KUKA KRL program: TORQUE.src

&ACCESS RV
&REL 9
&PARAM TEMPLATE = C:\KRC\Roboter\Template\FunctionVorgabe
&PARAM EDITMASK = *
DEFFCT BOOL TORQUE( )
DECL FRAME PT1
$TOOL=TOOL_DATA[5]
$ORI_TYPE=#CONSTANT
$VEL.CP=1.0
$VEL.ORI1=100
$VEL.ORI2=100
$ACC.CP=1.0
$ACC.ORI1=100
$ACC.ORI2=100

PTP $AXIS_ACT
IF $POS_ACT.A > 0 THEN
PTP_REL {A -1}
ENDIF
IF $POS_ACT.A < 0 THEN
PTP_REL {A 1}
ENDIF


ENDFCT
